TYPE DUT_MESSAGEFEED :
STRUCT
	ID: INT;
	Level: INT; //1:Success; 2:Info; 3:Warning; 4:ERROR; 5:FATAL
	Timestamp: STRING[80];
	Message: STRING[256];
END_STRUCT
END_TYPE

(* stored: Version 1.1.0.1, ProductVersion 3.1.0.25
   DUT DUT_MESSAGEFEED: Id {fab064d0-3aba-4dc1-aa5b-5bb1d44e5e03} *)
